// TIA Portal V19 export
DATA_BLOCK "DB_KorrPos"   // DB54
{ S7_Optimized_Access := 'FALSE' }
// stored: AutoNumber false
   VAR RETAIN
      Offset : Int := 10;   // Beginn erste Struktur
      Leng : Int := 200;   // Länge einer Struktur
      resI : Int := 0;
      Berechnung_ein : Bool := FALSE;   // * Berechnung durchführen
      res : Bool := FALSE;
      res1 : Bool := FALSE;
      res2 : Bool := FALSE;
      res3 : Bool := FALSE;
      res4 : Bool := FALSE;
      res5 : Bool := FALSE;
      res6 : Bool := FALSE;
      resB : Byte := 16#00;
      resI1 : Int := 0;
      TW : Array[1..10] of Struct
         Pos : Array[1..100] of Int;
      END_STRUCT;
   END_VAR
BEGIN
   TW[1].Pos[1..100] := 0;
   TW[2].Pos[1..100] := 0;
   TW[3].Pos[1..100] := 0;
   TW[4].Pos[1..100] := 0;
   TW[5].Pos[1..100] := 0;
   TW[6].Pos[1..100] := 0;
   TW[7].Pos[1..100] := 0;
   TW[8].Pos[1..100] := 0;
   TW[9].Pos[1..100] := 0;
   TW[10].Pos[1..100] := 0;
END_DATA_BLOCK
